{attribute 'qualified_only'}
{attribute 'strict'}
TYPE E_SafetyType :
(
	eSingleChannel := 0
);
END_TYPE

(* stored: Version 1.1.0.1, ProductVersion 3.1.4024.11
   DUT E_SafetyType: Id {31d145a3-5116-437d-829d-237f29d4bb04} *)
